FUNCTION_BLOCK FollowingCar
  (* Standard: 61499-2 *)
  (* Version 0.1, 2015-00-08, SYY, SYY-PC *)
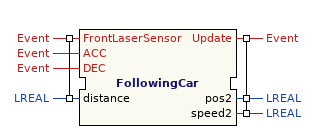
  EVENT_INPUT
    FrontLaserSensor WITH distance;
    ACC;
    DEC;
  END_EVENT
  EVENT_OUTPUT
    Update WITH pos2, speed2;
  END_EVENT
  VAR_INPUT
    distance : LREAL;
  END_VAR
  VAR_OUTPUT
    pos2 : LREAL := 0;
    speed2 : LREAL := 13.8;
  END_VAR
  VAR
    x : LREAL;
    v : LREAL;
    d : LREAL;
    k : INT;
    isInitial : BOOL;
    max : BOOL;
    min : BOOL;
  END_VAR
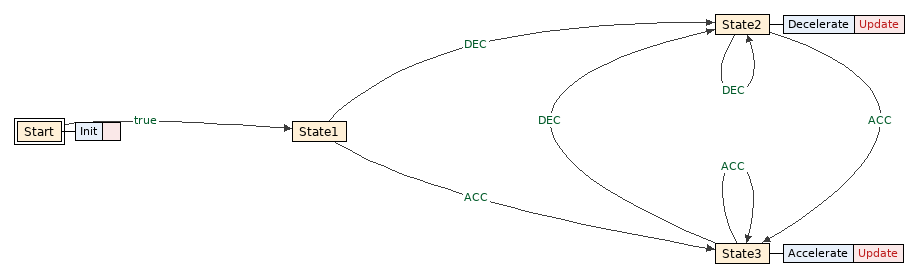
  EC_STATES
    Start : Init;
    State3 : Accelerate -> Update;
    State2 : Decelerate -> Update;
    State1;
  END_STATES
  EC_TRANSITIONS
    Start TO State1 := true;
    State3 TO State2 := DEC;
    State3 TO State3 := ACC;
    State2 TO State3 := ACC;
    State2 TO State2 := DEC;
    State1 TO State2 := DEC;
    State1 TO State3 := ACC;
  END_TRANSITIONS
  ALGORITHM Init IN C:
me->d = 0.01;
//me->v = 13.8;
me->speed2 = 13.8;
me->x = 0;
me->k = 366;
me->isInitial = true;
  END_ALGORITHM
  ALGORITHM Decelerate IN C:
me->v = me->speed2;
me->x = me->pos2;

//me->v = CarFollow_ode_1(C1v, d, k, s, x);
me->speed2 = me->v + me->d * 0.85 * (6.75 + 7.91 * tanh(0.13 * (me->distance - 5) - 1.57) - me->v);
me->pos2 = me->x + me->d * me->v;

printf("Following car decelerates (Position: %3.8f, Speed: %3.8f, Distance: %3.8f)\n", me->pos2, me->speed2, me->distance);
  END_ALGORITHM
  ALGORITHM Accelerate IN C:
me->v = me->speed2;
me->x = me->pos2;

//me->v = CarFollow_ode_1(C1v, d, k, s, x);
me->speed2 = me->v + me->d * 0.85 * (6.75 + 7.91 * tanh(0.13 * (me->distance - 5) - 1.57) - me->v);
me->pos2 = me->x + me->d * me->v;

printf("Following car accelerates (Position: %3.8f, Speed: %3.8f, Distance: %3.8f)\n", me->pos2, me->speed2, me->distance);
  END_ALGORITHM
  ALGORITHM Reset IN C:
if(!me->isInitial){
  me->k = 1;
}
  END_ALGORITHM
  ALGORITHM Init_Acc IN C:
me->max=false;
if(me->isInitial==false){
me->k = 0;
}
  END_ALGORITHM
  ALGORITHM Init_Dec IN C:
me->min=false;
if(me->isInitial==false){
me->k = 38;
}
  END_ALGORITHM
END_FUNCTION_BLOCK
